{attribute 'pack_mode' := '1'} //no gaps! (compiler tries to allign with base types and might skip bits otherwise)
{attribute 'analysis' := '-33'}
TYPE RbtFanucUnloadingt_DataOut_Grouped :
STRUCT
	_UI:RbtFanuc_ControlWord;			//24bits	>>start pt=1
	_DI:RbtFanucUnloading_DI;			//32 bits	>>start pt=25
	_GI:RbtFanucUnloading_GI;			//16 bits	>>start pt=57
END_STRUCT
END_TYPE

(* stored: Version 1.1.0.1
   DUT RbtFanucUnloadingt_DataOut_Grouped: Id {420222c1-9604-421c-bc36-925ea822a697} *)
